INTERFACE I_Logger EXTENDS I_FileProperties, I_HasAmsAddress

// Logs the message without any additions.
METHOD LogDefault
VAR_INPUT
	message	: Tc2_System.T_MaxString;
END_VAR
END_METHOD

END_INTERFACE

(* stored: Version 1.1.0.1, ProductVersion 3.1.4024.14
   Itf I_Logger: Id {8d645b62-749c-03d8-0193-52115f211da1}
   Method LogDefault: Id {a61e42ea-a189-0fbf-05f7-7abc3f7020f8} *)
